FUNCTION_BLOCK PUBLIC CannotCompareTypeError EXTENDS Error
VAR
	state : (CLEARED, RAISED);
	dataType1 : T_MAXSTRING;
	dataType2 : T_MAXSTRING;
END_VAR

PROPERTY Active : BOOL
GET
Active := state <> CLEARED;
END_GET
END_PROPERTY

METHOD PUBLIC Clear
dataType1 := '';
dataType2 := '';
state := CLEARED;
END_METHOD

PROPERTY PUBLIC ErrorCode : HRESULT
GET
ErrorCode := Tc2_System.E_HRESULTAdsErr.INCOMPATIBLE;
END_GET
END_PROPERTY

PROPERTY PUBLIC Message : T_MaxString
GET
Message := 'Cannot compare datatypes';
END_GET
END_PROPERTY

METHOD PUBLIC Raise
VAR_INPUT
	DataType1 : T_MAXSTRING;
	DataType2 : T_MAXSTRING;
END_VAR
THIS^.dataType1 := DataType1;
THIS^.dataType2 := DataType2;
state := RAISED;
END_METHOD

PROPERTY Reason : T_MaxString
GET
VAR
	message : STRING;
END_VAR
IF state = CLEARED THEN
	RETURN;
END_IF

message := CONCAT(message, dataType1);
message := CONCAT(message, ' with ');
message := CONCAT(message, dataType2);

Reason := message;
END_GET
END_PROPERTY

END_FUNCTION_BLOCK

(* stored: Version 1.1.0.1, ProductVersion 3.1.4024.12
   POU CannotCompareTypeError: Id {20ad30a3-ffe9-04b8-0a3b-f5bfd151bb67}, SpecialFunc None
   Property Active: Id {d0fc6167-f943-0d82-3d79-ae21b715b3a1}
   Get Get: Id {321841b4-b7c0-0b0c-3270-fd32ae1e2105}
   Method Clear: Id {a38ad8cc-90a2-09f0-3b8a-5efd1b85f959}
   Property ErrorCode: Id {02c83b7d-492d-0c72-0be7-506cd8c888d1}
   Get Get: Id {ca749e32-de49-0b0d-0f4d-8a170a8bc9e5}
   Property Message: Id {a19432c6-7047-0c39-0081-126df0120760}
   Get Get: Id {883c1809-31db-082b-027a-6cb77882c81a}
   Method Raise: Id {6355238d-9bca-0acd-0570-1a86c648189d}
   Property Reason: Id {8ccf31cc-fc88-02ca-3e10-a91176d3b285}
   Get Get: Id {b96fce93-9620-0ca4-2dc7-e1059408d91d} *)
